Universal Robots PolyScope program: SandCube.urp

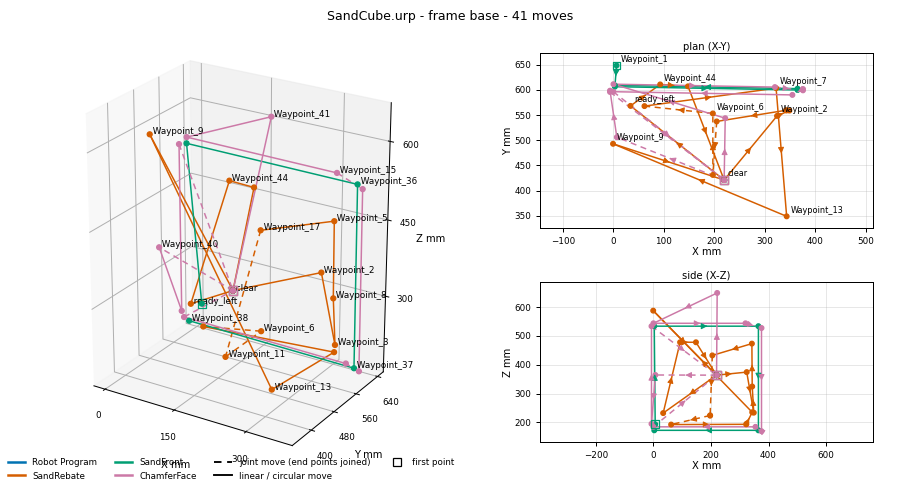
[picture p0: tool path of SandCube.urp in frame base, 41 of 41 moves have a stored position in this frame; points joined in program order, loops and branches not executed]
Program SandCube (installation=main2 directory=/programs createdIn=5.11.5.1010327 lastSavedIn=5.11.5.1010327 robotSerialNumber=20215500677)
Calibrated DH parameters: a=[0.000204, -0.239222, -0.391845, -0.000001, 0.000022, 0]; d=[0.162722, -355.808559, 353.37206, 2.570385, 0.099741, 0.099629]; alpha=[1.571124, 0.000988, 0.008295, 1.568963, -1.570303, 0]; deltaTheta=[0, -0.973091, 7.204745, 0.05153, 0, 0]
BeforeStart
  WorkPlane := CubeFront
Robot Program (runOnlyOnce=true)
  Folder Main
    MoveJ speed 60 deg/s, acceleration 80 deg/s^2 (useActiveTCP=false) tcp=DynabradeDual; feature=CubeFront
      Waypoint clear: TCP in base x=219.365 y=421.157 z=363.889 mm, rx=-1.5717 ry=-0.1089 rz=-0.0222 rad; joints [194.744, -106.958, 146.533, -122.37, 45.33, -106.867] deg; TCP offset x=3.18 y=114.64 z=98.2 mm, rx=-0.7854 ry=0 rz=0 rad; feature pose in base x=0.075 y=618.898 z=169.22 mm, rx=1.5781 ry=-0.0141 rz=-0.0141 rad
      URCap Zero FT Sensor (Robotiq_Copilot, Robotiq Inc.) dataModel(NodeInitializedKey=true, WaitForSteadyWrenchOptionKey=true)
  WorkPlane := CubeFront
  Call SandFront
  MoveJ speed 60 deg/s, acceleration 80 deg/s^2 (useActiveTCP=false) tcp=DynabradeDual; feature=CubeFront
    Waypoint clear: TCP in base x=219.365 y=421.157 z=363.889 mm, rx=-1.5717 ry=-0.1089 rz=-0.0222 rad; joints [194.744, -106.958, 146.533, -122.37, 45.33, -106.867] deg
    URCap Zero FT Sensor (Robotiq_Copilot, Robotiq Inc.) dataModel(NodeInitializedKey=true, WaitForSteadyWrenchOptionKey=true)
  Call ChamferFace
  MoveJ speed 60 deg/s, acceleration 80 deg/s^2 (useActiveTCP=false) tcp=DynabradeDual; feature=CubeFront
    Waypoint clear: TCP in base x=219.365 y=421.157 z=363.889 mm, rx=-1.5717 ry=-0.1089 rz=-0.0222 rad; joints [194.744, -106.958, 146.533, -122.37, 45.33, -106.867] deg
    URCap Zero FT Sensor (Robotiq_Copilot, Robotiq Inc.) dataModel(NodeInitializedKey=true, WaitForSteadyWrenchOptionKey=true)
  WorkPlane := SandBack
  MoveJ speed 60 deg/s, acceleration 80 deg/s^2 (useActiveTCP=false) tcp=DynabradeDual; feature=SandBack
    Waypoint clear: TCP in base x=219.365 y=421.157 z=363.889 mm, rx=-1.5717 ry=-0.1089 rz=-0.0222 rad; joints [194.744, -106.958, 146.533, -122.37, 45.33, -106.867] deg
    URCap Zero FT Sensor (Robotiq_Copilot, Robotiq Inc.) dataModel(NodeInitializedKey=true, WaitForSteadyWrenchOptionKey=true)
  Call SandFront
  MoveJ speed 60 deg/s, acceleration 80 deg/s^2 (useActiveTCP=false) tcp=DynabradeDual; feature=SandBack
    Waypoint clear: TCP in base x=219.365 y=421.157 z=363.889 mm, rx=-1.5717 ry=-0.1089 rz=-0.0222 rad; joints [194.744, -106.958, 146.533, -122.37, 45.33, -106.867] deg
    URCap Zero FT Sensor (Robotiq_Copilot, Robotiq Inc.) dataModel(NodeInitializedKey=true, WaitForSteadyWrenchOptionKey=true)
  Call ChamferFace
  MoveJ speed 60 deg/s, acceleration 80 deg/s^2 (useActiveTCP=false) tcp=DynabradeDual; feature=SandBack
    Waypoint clear: TCP in base x=219.365 y=421.157 z=363.889 mm, rx=-1.5717 ry=-0.1089 rz=-0.0222 rad; joints [194.744, -106.958, 146.533, -122.37, 45.33, -106.867] deg
    URCap Zero FT Sensor (Robotiq_Copilot, Robotiq Inc.) dataModel(NodeInitializedKey=true, WaitForSteadyWrenchOptionKey=true)
SubProgram -> ChamferFace
Event  expression=digital_in[1]≠ True
  Set DigitalOutput pin=digital_out[0]; digitalValue=0
  Set DigitalOutput pin=digital_out[1]; digitalValue=0
  Halt
SubProgram SandRebate (keepSynchronizedWithDisk=false)
  Folder sandRebate
    MoveJ speed 60 deg/s, acceleration 80 deg/s^2 (useActiveTCP=false) tcp=DynabradeDual; feature=CubeFront
      Waypoint clear: TCP in base x=219.365 y=421.157 z=363.889 mm, rx=-1.5717 ry=-0.1089 rz=-0.0222 rad; joints [194.744, -106.958, 146.533, -122.37, 45.33, -106.867] deg
      URCap Zero FT Sensor (Robotiq_Copilot, Robotiq Inc.) dataModel(NodeInitializedKey=true, WaitForSteadyWrenchOptionKey=true)
      MoveL speed 250 mm/s, acceleration 1200 mm/s^2 (useActiveTCP=false) tcp=DynabradeDual; feature=CubeFront
        Waypoint ready_left: TCP in base x=33.773 y=568.14 z=232.075 mm, rx=-1.2213 ry=-1.2022 rz=1.1979 rad; joints [233.005, -43.676, 101.374, -178.142, 55.004, -44.435] deg; TCP offset x=3.18 y=114.64 z=98.2 mm, rx=-0.7854 ry=0 rz=0 rad; feature pose in base x=9.685 y=618.378 z=176.869 mm, rx=1.5687 ry=-0.014 rz=-0.0074 rad
        URCap Find Surface (Robotiq_Copilot, Robotiq Inc.) dataModel(NodeInitializedKey=true, WaitForSteadyWrenchOptionKey=false, ls_force=10.0, ls_distance=100.0, ls_speed=5.0, ZeroSensorBeforeKey=true, ls_if_distance=false, ls_if_force=false); state(isChildrenLocked=true)
          'Add Stop conditions from the Find Surface node'
        URCap Finishing Tool Control (Robotiq_Copilot, Robotiq Inc.) dataModel(ToolOutputNameKey=digital_out[0], HackTriggeringContributionIsDefinedMethodKey=true)
        Wait Sleep waitTime=0.5
        Force Simple feature=Joint_6_name; selection=[0, 0, 1, 0, 0, 0]; wrench=[0, 0, 5, 0, 0, 0]; limitsForce=[0.15, 0.15, 0.15, 1.047198, 1.047198, 1.047198]; limitsMotion=[0.1, 0.1, 0.1, 0.349066, 0.349066, 0.349066]
          Waypoint Waypoint_44: motionParameters(jointSpeed=1.047198 jointAcceleration=1.396263 cartesianSpeed=0.05 cartesianAcceleration=1.2); TCP in base x=92.634 y=610.628 z=478.238 mm, rx=-0.8396 ry=-1.4025 rz=0.8393 rad; joints [232.816, -51.553, 73.036, -159.375, 69.035, -55.707] deg; TCP offset x=3.18 y=114.64 z=98.2 mm, rx=-0.7854 ry=0 rz=0 rad; feature pose in base x=85.344 y=655.608 z=190.328 mm, rx=1.5707 ry=0.001 rz=-0.0012 rad
        URCap Finishing Tool Control (Robotiq_Copilot, Robotiq Inc.) dataModel(ToolOutputNameKey=digital_out[0], HackTriggeringContributionIsDefinedMethodKey=true, FinishingToolStateKey=false)
        Waypoint Waypoint_4: TCP in base x=147.72 y=606.874 z=478.224 mm, rx=-0.8396 ry=-1.4025 rz=0.8394 rad; joints [229.161, -48.232, 67.407, -157.963, 71.791, -53.121] deg
        Waypoint clear: TCP in base x=219.365 y=421.157 z=363.889 mm, rx=-1.5717 ry=-0.1089 rz=-0.0222 rad; joints [194.744, -106.958, 146.533, -122.37, 45.33, -106.867] deg; feature pose in base x=0.075 y=618.898 z=169.22 mm, rx=1.5781 ry=-0.0141 rz=-0.0141 rad
        Waypoint Waypoint_2: TCP in base x=324.212 y=548.214 z=374.491 mm, rx=-1.2092 ry=1.2092 rz=-1.2092 rad; joints [245.591, -72.937, 106.11, -100.873, 130.52, -237.51] deg; feature pose in base x=6.058 y=653.089 z=192.929 mm, rx=1.5716 ry=0.003 rz=-0.0025 rad
        Waypoint Waypoint_3: TCP in base x=348.673 y=558.868 z=233.4 mm, rx=-1.199 ry=1.2125 rz=-1.2251 rad; joints [243.834, -57.283, 109.058, -119.037, 129.688, -236.76] deg; TCP offset x=3.18 y=114.64 z=98.2 mm, rx=-0.7854 ry=0 rz=0 rad; feature pose in base x=9.685 y=618.378 z=176.869 mm, rx=1.5687 ry=-0.014 rz=-0.0074 rad
        URCap Find Surface (Robotiq_Copilot, Robotiq Inc.) dataModel(NodeInitializedKey=true, WaitForSteadyWrenchOptionKey=false, ls_force=10.0, ls_distance=100.0, ls_speed=5.0, ls_if_distance=false, ls_if_force=false, ZeroSensorBeforeKey=true); state(isChildrenLocked=true)
          'Add Stop conditions from the Find Surface node'
        URCap Finishing Tool Control (Robotiq_Copilot, Robotiq Inc.) dataModel(ToolOutputNameKey=digital_out[0], HackTriggeringContributionIsDefinedMethodKey=true)
        Wait Sleep waitTime=0.5
        Force Simple feature=Joint_6_name; selection=[0, 0, 1, 0, 0, 0]; wrench=[0, 0, 5, 0, 0, 0]; limitsForce=[0.15, 0.15, 0.15, 1.047198, 1.047198, 1.047198]; limitsMotion=[0.1, 0.1, 0.1, 0.349066, 0.349066, 0.349066]
          Waypoint Waypoint_8: motionParameters(jointSpeed=1.047198 jointAcceleration=1.396263 cartesianSpeed=0.05 cartesianAcceleration=1.2); TCP in base x=343.269 y=559.127 z=324.456 mm, rx=2.2046 ry=-0.0122 rz=2.2215 rad; joints [241.547, -71.33, 93.008, -21.809, 107.451, -270.149] deg; TCP offset x=3.18 y=114.64 z=98.2 mm, rx=-0.7854 ry=0 rz=0 rad
          Waypoint Waypoint_5: motionParameters(jointSpeed=1.047198 jointAcceleration=1.396263 cartesianSpeed=0.05 cartesianAcceleration=1.2); TCP in base x=342.13 y=559.447 z=473.527 mm, rx=2.1002 ry=0.2016 rz=2.1132 rad; joints [241.727, -73.096, 71.489, 10.077, 107.843, -275.731] deg; TCP offset x=3.18 y=114.64 z=98.2 mm, rx=-0.7854 ry=0 rz=0 rad
        URCap Finishing Tool Control (Robotiq_Copilot, Robotiq Inc.) dataModel(FinishingToolStateKey=false, ToolOutputNameKey=digital_out[0], HackTriggeringContributionIsDefinedMethodKey=true)
        Waypoint Waypoint_17: TCP in base x=204.615 y=537.314 z=432.533 mm, rx=-1.1836 ry=-1.1482 rz=-1.3158 rad; joints [212.134, -87.867, 98.846, 1.992, -9.504, -287.219] deg; TCP offset x=3.18 y=114.64 z=98.2 mm, rx=-0.7854 ry=0 rz=0 rad; feature pose in base x=6.058 y=653.089 z=192.929 mm, rx=1.5716 ry=0.003 rz=-0.0025 rad
        MoveJ speed 60 deg/s, acceleration 80 deg/s^2 (useActiveTCP=true) feature=CubeFront
          Waypoint Waypoint_11: TCP in base x=197.023 y=431.256 z=223.624 mm, rx=2.362 ry=2.0713 rz=0 rad; joints [223.025, -89.028, 102.064, -70.501, -56.519, -139.472] deg
          Waypoint Waypoint_6: TCP in base x=196.959 y=553.123 z=223.756 mm, rx=-1.75 ry=-2.609 rz=-0.0001 rad; joints [233.913, -69.804, 77.285, -56.958, -67.897, -156.703] deg
          Waypoint Waypoint_31: TCP in base x=61.467 y=567.687 z=192.19 mm, rx=1.7638 ry=2.5902 rz=0.0029 rad; joints [245.976, -73.297, 87.687, -68.963, -60.284, -145.062] deg; TCP offset x=3.18 y=114.64 z=98.2 mm, rx=-0.7854 ry=0 rz=0 rad; feature pose in base x=9.685 y=618.378 z=176.869 mm, rx=1.5687 ry=-0.014 rz=-0.0074 rad
          URCap Zero FT Sensor (Robotiq_Copilot, Robotiq Inc.) dataModel(NodeInitializedKey=true, WaitForSteadyWrenchOptionKey=true)
        URCap Find Surface (Robotiq_Copilot, Robotiq Inc.) dataModel(NodeInitializedKey=true, ZeroSensorBeforeKey=true, WaitForSteadyWrenchOptionKey=false, ls_force=10.0, ls_distance=100.0, ls_speed=5.0, ls_if_distance=false, ls_if_force=false); state(isChildrenLocked=true)
          'Add Stop conditions from the Find Surface node'
        URCap Finishing Tool Control (Robotiq_Copilot, Robotiq Inc.) dataModel(ToolOutputNameKey=digital_out[0], HackTriggeringContributionIsDefinedMethodKey=true)
        Wait Sleep waitTime=0.5
        Force Frame feature=Joint_6_name; selection=[0, 0, 1, 0, 0, 0]; wrench=[0, 0, 5, 0, 0, 0]; limitsForce=[0.15, 0.15, 0.15, 1.047198, 1.047198, 1.047198]; limitsMotion=[0.1, 0.1, 0.1, 0.349066, 0.349066, 0.349066]
          Waypoint Waypoint_7: motionParameters(jointSpeed=1.047198 jointAcceleration=1.396263 cartesianSpeed=0.05 cartesianAcceleration=1.2); TCP in base x=322.305 y=603.203 z=193.01 mm, rx=2.5491 ry=1.8349 rz=-0.0035 rad; joints [225.958, -61.111, 72.887, -78.246, -49.944, -124.133] deg; TCP offset x=3.18 y=114.64 z=98.2 mm, rx=-0.7854 ry=0 rz=0 rad; feature pose in base x=6.058 y=653.089 z=192.929 mm, rx=1.5716 ry=0.003 rz=-0.0025 rad
        URCap Finishing Tool Control (Robotiq_Copilot, Robotiq Inc.) dataModel(FinishingToolStateKey=false, ToolOutputNameKey=digital_out[0], HackTriggeringContributionIsDefinedMethodKey=true)
        Waypoint Waypoint_13: TCP in base x=343.245 y=349.195 z=234.967 mm, rx=-1.8514 ry=-2.5381 rz=0.0001 rad; joints [208.052, -81.166, 89.339, -53.576, -82.434, -172.912] deg; feature pose in base x=9.685 y=618.378 z=176.869 mm, rx=1.5687 ry=-0.014 rz=-0.0074 rad
        Waypoint Waypoint_9: TCP in base x=-0.811 y=492.962 z=588.061 mm, rx=-1.9827 ry=-0.1778 rz=-0.0774 rad; joints [237.765, -113.533, 89.133, -2.101, 52.621, -171.272] deg
        Waypoint clear: TCP in base x=219.365 y=421.157 z=363.889 mm, rx=-1.5717 ry=-0.1089 rz=-0.0222 rad; joints [194.744, -106.958, 146.533, -122.37, 45.33, -106.867] deg; feature pose in base x=0.075 y=618.898 z=169.22 mm, rx=1.5781 ry=-0.0141 rz=-0.0141 rad
SubProgram SprayFront [hidden by the author, left out]
SubProgram SprayRebate [hidden by the author, left out]
SubProgram -> SandFront
SubProgram StartSpray [hidden by the author, left out]
SubProgram stopSpray [hidden by the author, left out]
SubProgram SandFront (keepSynchronizedWithDisk=false)
  Folder sandFront
    MoveL speed 250 mm/s, acceleration 1200 mm/s^2 (useActiveTCP=false) tcp=DynabradeDual; feature=WorkPlane
      Waypoint Waypoint_1: TCP in base x=6.072 y=648.1 z=192.982 mm, rx=-1.5699 ry=0.0092 rz=0.0097 rad; joints [251.403, -67.593, 131.535, -110.394, 77.851, -166.352] deg; feature pose in base x=6.058 y=653.089 z=192.929 mm, rx=1.5716 ry=0.003 rz=-0.0025 rad
      URCap Zero FT Sensor (Robotiq_Copilot, Robotiq Inc.) dataModel(NodeInitializedKey=true, WaitForSteadyWrenchOptionKey=true)
      URCap Find Surface (Robotiq_Copilot, Robotiq Inc.) dataModel(NodeInitializedKey=true, WaitForSteadyWrenchOptionKey=false, ls_force=10.0, ls_distance=100.0, ls_speed=5.0, ZeroSensorBeforeKey=false, ls_if_distance=false, ls_if_force=false); state(isChildrenLocked=true)
        'Add Stop conditions from the Find Surface node'
      URCap Finishing Tool Control (Robotiq_Copilot, Robotiq Inc.) dataModel(ToolOutputNameKey=digital_out[0], HackTriggeringContributionIsDefinedMethodKey=true)
      Wait Sleep waitTime=0.5
    MoveL speed 60 mm/s, acceleration 1200 mm/s^2 (useActiveTCP=false) tcp=DynabradeDual; feature=WorkPlane
      Force Simple feature=Joint_6_name; selection=[0, 0, 1, 0, 0, 0]; wrench=[0, 0, 5, 0, 0, 0]; limitsForce=[0.15, 0.15, 0.15, 1.047198, 1.047198, 1.047198]; limitsMotion=[0.1, 0.1, 0.1, 0.349066, 0.349066, 0.349066]
        Waypoint Waypoint_35: TCP in base x=2.83 y=606.158 z=534.136 mm, rx=-1.5633 ry=0.0141 rz=-0.0141 rad; joints [250.421, -103.852, 108.643, -51.818, 77.42, -166.342] deg; TCP offset x=3.18 y=114.64 z=98.2 mm, rx=-0.7854 ry=0 rz=0 rad; feature pose in base x=0.075 y=618.898 z=169.22 mm, rx=1.5781 ry=-0.0141 rz=-0.0141 rad
        Waypoint Waypoint_36: TCP in base x=364.819 y=599.647 z=534.105 mm, rx=-1.5633 ry=0.0141 rz=-0.0141 rad; joints [211.846, -86.054, 95.624, -71.528, 54.288, -132.089] deg; TCP offset x=3.18 y=114.64 z=98.2 mm, rx=-0.7854 ry=0 rz=0 rad
        Waypoint Waypoint_37: TCP in base x=364.836 y=602.311 z=172.118 mm, rx=-1.5633 ry=0.0141 rz=-0.0141 rad; joints [212.02, -54.973, 118.464, -125.048, 54.344, -132.771] deg; TCP offset x=3.18 y=114.64 z=98.2 mm, rx=-0.7854 ry=0 rz=0 rad
        Waypoint Waypoint_38: TCP in base x=2.894 y=608.811 z=172.149 mm, rx=-1.5633 ry=0.0141 rz=-0.0141 rad; joints [250.409, -66.525, 138.189, -118.584, 77.481, -166.829] deg; TCP offset x=3.18 y=114.64 z=98.2 mm, rx=-0.7854 ry=0 rz=0 rad
        URCap Finishing Tool Control (Robotiq_Copilot, Robotiq Inc.) dataModel(FinishingToolStateKey=false, ToolOutputNameKey=digital_out[0], HackTriggeringContributionIsDefinedMethodKey=true)
      MoveDirectionNode (selectedDirection=ZMinus) feature=Joint_6_name
        Until DISTANCE (allowActions=false deceleration=3 distanceNodeType=STOP) Distance=0.025; motionParameters(blendRadius=0)
SubProgram ChamferFace (keepSynchronizedWithDisk=false)
  SuppressedNode
    WorkPlane := SandBack
  MoveJ speed 60 deg/s, acceleration 80 deg/s^2 (useActiveTCP=false) tcp=DynabradeDual; feature=WorkPlane
    Waypoint clear: TCP in base x=219.365 y=421.157 z=363.889 mm, rx=-1.5717 ry=-0.1089 rz=-0.0222 rad; joints [194.744, -106.958, 146.533, -122.37, 45.33, -106.867] deg; TCP offset x=3.18 y=114.64 z=98.2 mm, rx=-0.7854 ry=0 rz=0 rad
    MoveL speed 250 mm/s, acceleration 1200 mm/s^2 (useActiveTCP=true) feature=WorkPlane
      Waypoint Waypoint_41: TCP in base x=221.5 y=543.735 z=649.649 mm, rx=-1.5717 ry=-0.1089 rz=-0.022 rad; joints [214.426, -103.918, 95.357, -57.203, 50.729, -131.892] deg
      Waypoint Waypoint_14: TCP in base x=-0.008 y=611.132 z=544.162 mm, rx=-2.3487 ry=0.0212 rz=-0.0088 rad; joints [252.136, -85.085, 59.128, 25.398, 72.909, -179.557] deg
    URCap Find Surface (Robotiq_Copilot, Robotiq Inc.) dataModel(NodeInitializedKey=true, WaitForSteadyWrenchOptionKey=false, ls_force=10.0, ls_distance=100.0, ls_speed=5.0, ZeroSensorBeforeKey=true, ls_if_distance=false, ls_if_force=false); state(isChildrenLocked=true)
      'Add Stop conditions from the Find Surface node'
    URCap Finishing Tool Control (Robotiq_Copilot, Robotiq Inc.) dataModel(ToolOutputNameKey=digital_out[0], HackTriggeringContributionIsDefinedMethodKey=true)
    Wait Sleep waitTime=1
    Force Simple feature=Joint_6_name; selection=[0, 0, 1, 0, 0, 0]; wrench=[0, 0, 2, 0, 0, 0]; limitsForce=[0.15, 0.15, 0.15, 1.047198, 1.047198, 1.047198]; limitsMotion=[0.1, 0.1, 0.1, 0.349066, 0.349066, 0.349066]
      MoveL speed 250 mm/s, acceleration 1200 mm/s^2 (useActiveTCP=false) tcp=DynabradeDual; feature=WorkPlane
        Waypoint Waypoint_15: TCP in base x=319.916 y=605.399 z=544.112 mm, rx=-2.3488 ry=0.0213 rz=-0.0087 rad; joints [217.403, -68.511, 37.925, 29.506, 38.137, -178.971] deg; TCP offset x=3.18 y=114.64 z=98.2 mm, rx=-0.7854 ry=0 rz=0 rad
        URCap Finishing Tool Control (Robotiq_Copilot, Robotiq Inc.) dataModel(FinishingToolStateKey=false, ToolOutputNameKey=digital_out[0], HackTriggeringContributionIsDefinedMethodKey=true)
    MoveL speed 250 mm/s, acceleration 1200 mm/s^2 (useActiveTCP=false) tcp=DynabradeDual; feature=WorkPlane
      MoveDirectionNode (selectedDirection=ZMinus) feature=Joint_6_name
        Until DISTANCE (allowActions=false deceleration=3 distanceNodeType=STOP) Distance=0.1; motionParameters(blendRadius=0)
    MoveJ speed 60 deg/s, acceleration 80 deg/s^2 (useActiveTCP=false) tcp=DynabradeDual; feature=WorkPlane
      Waypoint Waypoint_16: TCP in base x=375.551 y=598.897 z=527.773 mm, rx=-1.7433 ry=0.7352 rz=1.7487 rad; joints [207.169, -56.155, 39.199, 15.353, 27.996, -88.419] deg; TCP offset x=3.18 y=114.64 z=98.2 mm, rx=-0.7854 ry=0 rz=0 rad
      URCap Find Surface (Robotiq_Copilot, Robotiq Inc.) dataModel(NodeInitializedKey=true, WaitForSteadyWrenchOptionKey=false, ls_force=10.0, ls_distance=100.0, ls_speed=5.0, ZeroSensorBeforeKey=true, ls_if_distance=false, ls_if_force=false); state(isChildrenLocked=true)
        'Add Stop conditions from the Find Surface node'
      URCap Finishing Tool Control (Robotiq_Copilot, Robotiq Inc.) dataModel(ToolOutputNameKey=digital_out[0], HackTriggeringContributionIsDefinedMethodKey=true)
      Wait Sleep waitTime=1
      Force Simple feature=Joint_6_name; selection=[0, 0, 1, 0, 0, 0]; wrench=[0, 0, 2, 0, 0, 0]; limitsForce=[0.15, 0.15, 0.15, 1.047198, 1.047198, 1.047198]; limitsMotion=[0.1, 0.1, 0.1, 0.349066, 0.349066, 0.349066]
        MoveL speed 250 mm/s, acceleration 1200 mm/s^2 (useActiveTCP=false) tcp=DynabradeDual; feature=WorkPlane
          Waypoint Waypoint_18: TCP in base x=375.596 y=601.544 z=169.103 mm, rx=-1.7433 ry=0.7352 rz=1.7487 rad; joints [207.38, -48.328, 80.471, -33.664, 28.599, -88.508] deg
          URCap Finishing Tool Control (Robotiq_Copilot, Robotiq Inc.) dataModel(FinishingToolStateKey=false, ToolOutputNameKey=digital_out[0], HackTriggeringContributionIsDefinedMethodKey=true)
      MoveL speed 250 mm/s, acceleration 1200 mm/s^2 (useActiveTCP=false) tcp=DynabradeDual; feature=WorkPlane
        MoveDirectionNode (selectedDirection=ZMinus) feature=Joint_6_name
          Until DISTANCE (allowActions=false deceleration=3 distanceNodeType=STOP) Distance=0.15; motionParameters(blendRadius=0)
    MoveJ speed 60 deg/s, acceleration 80 deg/s^2 (useActiveTCP=false) tcp=DynabradeDual; feature=WorkPlane
      Waypoint Waypoint_19: TCP in base x=354.585 y=589.87 z=184.268 mm, rx=-0.6415 ry=0.6531 rz=1.455 rad; joints [220.483, -48.221, 112.687, -93.081, 94.888, -59.639] deg; TCP offset x=3.18 y=114.64 z=98.2 mm, rx=-0.7854 ry=0 rz=0 rad
      URCap Find Surface (Robotiq_Copilot, Robotiq Inc.) dataModel(NodeInitializedKey=true, WaitForSteadyWrenchOptionKey=false, ls_force=10.0, ls_distance=100.0, ls_speed=5.0, ZeroSensorBeforeKey=true, ls_if_distance=false, ls_if_force=false); state(isChildrenLocked=true)
        'Add Stop conditions from the Find Surface node'
      URCap Finishing Tool Control (Robotiq_Copilot, Robotiq Inc.) dataModel(ToolOutputNameKey=digital_out[0], HackTriggeringContributionIsDefinedMethodKey=true)
      Wait Sleep waitTime=1
      Force Simple feature=Joint_6_name; selection=[0, 0, 1, 0, 0, 0]; wrench=[0, 0, 2, 0, 0, 0]; limitsForce=[0.15, 0.15, 0.15, 1.047198, 1.047198, 1.047198]; limitsMotion=[0.1, 0.1, 0.1, 0.349066, 0.349066, 0.349066]
        MoveL speed 250 mm/s, acceleration 1200 mm/s^2 (useActiveTCP=false) tcp=DynabradeDual; feature=WorkPlane
          Waypoint Waypoint_20: TCP in base x=-0.331 y=596.237 z=184.279 mm, rx=-0.6415 ry=0.6532 rz=1.455 rad; joints [260.295, -52.025, 128.164, -113.807, 128.741, -82.873] deg; TCP offset x=3.18 y=114.64 z=98.2 mm, rx=-0.7854 ry=0 rz=0 rad
          URCap Finishing Tool Control (Robotiq_Copilot, Robotiq Inc.) dataModel(FinishingToolStateKey=false, ToolOutputNameKey=digital_out[0], HackTriggeringContributionIsDefinedMethodKey=true)
      MoveL speed 250 mm/s, acceleration 1200 mm/s^2 (useActiveTCP=false) tcp=DynabradeDual; feature=WorkPlane
        MoveDirectionNode (selectedDirection=ZMinus) feature=Joint_6_name
          Until DISTANCE (allowActions=false deceleration=3 distanceNodeType=STOP) Distance=0.15; motionParameters(blendRadius=0)
    MoveJ speed 60 deg/s, acceleration 80 deg/s^2 (useActiveTCP=false) tcp=DynabradeDual; feature=WorkPlane
      Waypoint clear: TCP in base x=219.365 y=421.157 z=363.889 mm, rx=-1.5717 ry=-0.1089 rz=-0.0222 rad; joints [194.744, -106.958, 146.533, -122.37, 45.33, -106.867] deg; TCP offset x=3.18 y=114.64 z=98.2 mm, rx=-0.7854 ry=0 rz=0 rad
      Waypoint Waypoint_40: TCP in base x=6.663 y=506.081 z=364.462 mm, rx=-1.5718 ry=-0.1088 rz=-0.022 rad; joints [237.975, -113.969, 141.657, -79.771, 63.213, -156.294] deg
    MoveL speed 250 mm/s, acceleration 1200 mm/s^2 (useActiveTCP=false) tcp=DynabradeDual; feature=WorkPlane
      Waypoint Waypoint_34: TCP in base x=-6.831 y=598.251 z=194.775 mm, rx=-1.7669 ry=-0.7078 rz=-1.7722 rad; joints [268.715, -45.999, 120.301, -254.699, -90.143, -89.729] deg
      URCap Find Surface (Robotiq_Copilot, Robotiq Inc.) dataModel(NodeInitializedKey=true, WaitForSteadyWrenchOptionKey=false, ls_force=10.0, ls_distance=100.0, ls_speed=5.0, ZeroSensorBeforeKey=true, ls_if_distance=false, ls_if_force=false); state(isChildrenLocked=true)
        'Add Stop conditions from the Find Surface node'
      URCap Finishing Tool Control (Robotiq_Copilot, Robotiq Inc.) dataModel(ToolOutputNameKey=digital_out[0], HackTriggeringContributionIsDefinedMethodKey=true)
      Wait Sleep waitTime=1
      Force Simple feature=Joint_6_name; selection=[0, 0, 1, 0, 0, 0]; wrench=[0, 0, 2, 0, 0, 0]; limitsForce=[0.15, 0.15, 0.15, 1.047198, 1.047198, 1.047198]; limitsMotion=[0.1, 0.1, 0.1, 0.349066, 0.349066, 0.349066]
        MoveL speed 250 mm/s, acceleration 1200 mm/s^2 (useActiveTCP=false) tcp=DynabradeDual; feature=WorkPlane
          Waypoint Waypoint_39: TCP in base x=-6.825 y=595.748 z=534.059 mm, rx=-1.767 ry=-0.7079 rz=-1.7723 rad; joints [268.636, -84.886, 108.224, -203.734, -89.802, -89.466] deg; TCP offset x=3.18 y=114.64 z=98.2 mm, rx=-0.7854 ry=0 rz=0 rad
          URCap Finishing Tool Control (Robotiq_Copilot, Robotiq Inc.) dataModel(FinishingToolStateKey=false, ToolOutputNameKey=digital_out[0], HackTriggeringContributionIsDefinedMethodKey=true)
      MoveL speed 250 mm/s, acceleration 1200 mm/s^2 (useActiveTCP=false) tcp=DynabradeDual; feature=WorkPlane
        MoveDirectionNode (selectedDirection=ZMinus) feature=Joint_6_name
          Until DISTANCE (allowActions=false deceleration=3 distanceNodeType=STOP) Distance=0.15; motionParameters(blendRadius=0)
    MoveJ speed 60 deg/s, acceleration 80 deg/s^2 (useActiveTCP=false) tcp=DynabradeDual; feature=WorkPlane
      Waypoint clear: TCP in base x=219.365 y=421.157 z=363.889 mm, rx=-1.5717 ry=-0.1089 rz=-0.0222 rad; joints [194.744, -106.958, 146.533, -122.37, 45.33, -106.867] deg; TCP offset x=3.18 y=114.64 z=98.2 mm, rx=-0.7854 ry=0 rz=0 rad
